Staubli VAL3: fitCircle.pgx

program fitCircle()
begin
  //fit a circle through pPointIn array.
  nCircleErr=$circleFind(pPointIn,fCircleFrame,nRadius)
  if nCircleErr<0
    gotoxy(1,10)
    put("圆:拟合失败！")
    return
  endIf
  gotoxy(1,10)
  put("圆半径："+toString(".2",nRadius)+"  "+"误差："+toString(".2",nCircleErr))
end
